TYPE ST_LinearPumpCalibration :
STRUCT
	bEnabled 		: BOOL;
	bHomed			: BOOL;
	rOldPosition	: LREAL;
	rNewPosition	: LREAL;
	bActivate		: BOOL;
END_STRUCT
END_TYPE

(* stored: Version 1.1.0.1, ProductVersion 3.1.4024.12
   DUT ST_LinearPumpCalibration: Id {4426d1db-f74d-43a3-b2be-0760eb24c42e} *)
